SUBAPPLICATION Uebung_039 (* Spiegelabfolge V2 mit Schrittkette *)
  (* Standard: 61499-2; Description: Spiegelabfolge V2 mit Schrittkette geeignet für hydraulische 4/3 Wege Ventile oder pneumatische 5/3 Wege Ventile jeweils Mittelstellung gesperrt. *)
  (* Version 1.0, 2023-10-23, franz *)
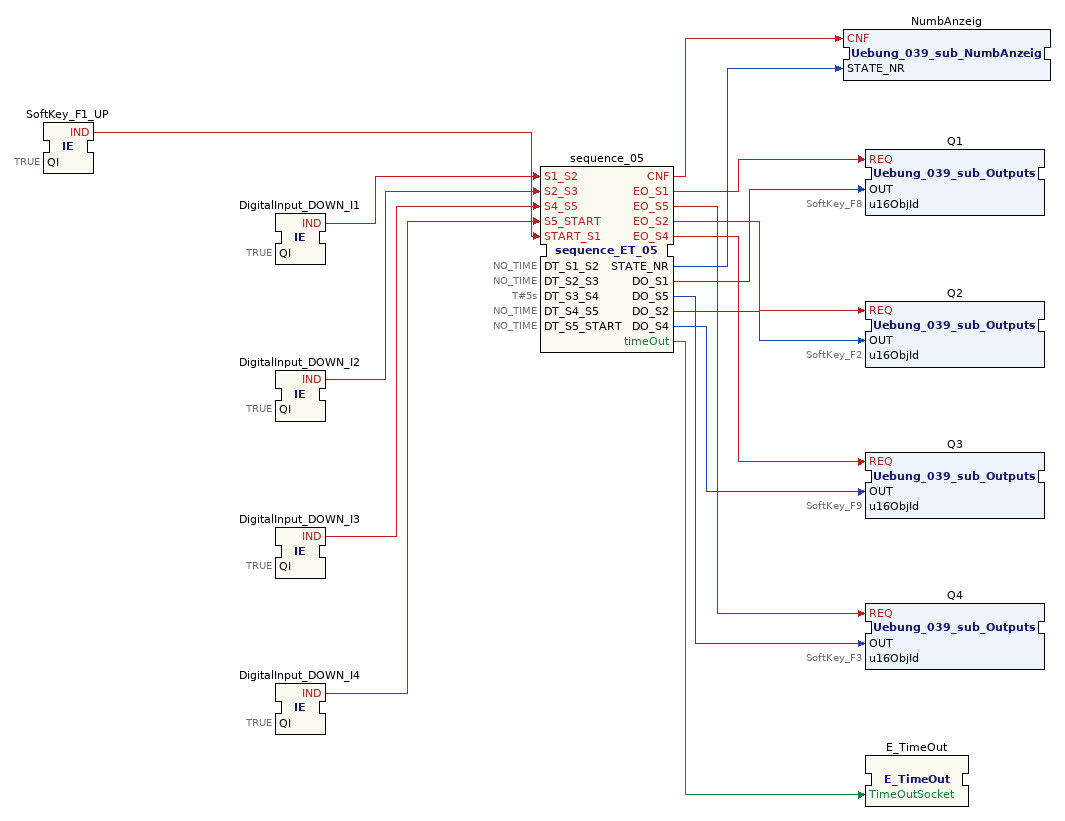
  FBS
    E_TimeOut : E_TimeOut;
    DigitalInput_DOWN_I1 : IE(QI := TRUE);
    DigitalInput_DOWN_I2 : IE(QI := TRUE);
    DigitalInput_DOWN_I3 : IE(QI := TRUE);
    DigitalInput_DOWN_I4 : IE(QI := TRUE);
    sequence_05 : sequence_ET_05(DT_S1_S2 := NO_TIME, DT_S2_S3 := NO_TIME, DT_S3_S4 := T#5s, DT_S4_S5 := NO_TIME, DT_S5_START := NO_TIME);
    SoftKey_F1_UP : IE(QI := TRUE);
  END_FBS
  SUBAPPS
    NumbAnzeig : Uebung_039_sub_NumbAnzeig;
    Q1 : Uebung_039_sub_Outputs(u16ObjId := SoftKey_F8);
    Q4 : Uebung_039_sub_Outputs(u16ObjId := SoftKey_F3);
    Q2 : Uebung_039_sub_Outputs(u16ObjId := SoftKey_F2);
    Q3 : Uebung_039_sub_Outputs(u16ObjId := SoftKey_F9);
  END_SUBAPPS
  EVENT_CONNECTIONS
    DigitalInput_DOWN_I1.IND TO sequence_05.S1_S2;
    DigitalInput_DOWN_I2.IND TO sequence_05.S2_S3;
    DigitalInput_DOWN_I3.IND TO sequence_05.S4_S5;
    DigitalInput_DOWN_I4.IND TO sequence_05.S5_START;
    sequence_05.CNF TO NumbAnzeig.CNF;
    SoftKey_F1_UP.IND TO sequence_05.START_S1;
    sequence_05.EO_S1 TO Q1.REQ;
    sequence_05.EO_S5 TO Q4.REQ;
    sequence_05.EO_S2 TO Q2.REQ;
    sequence_05.EO_S4 TO Q3.REQ;
  END_CONNECTIONS
  DATA_CONNECTIONS
    sequence_05.STATE_NR TO NumbAnzeig.STATE_NR;
    sequence_05.DO_S1 TO Q1.OUT;
    sequence_05.DO_S5 TO Q4.OUT;
    sequence_05.DO_S2 TO Q2.OUT;
    sequence_05.DO_S4 TO Q3.OUT;
  END_CONNECTIONS
  ADAPTER_CONNECTIONS
    sequence_05.timeOut TO E_TimeOut.TimeOutSocket;
  END_CONNECTIONS
END_SUBAPPLICATION
